{attribute addProperty BoxType "EL6022-0000-0016"}
{attribute addProperty Id "COM_Inputs_ChannelAT %I*ARRAY[0..1] OF COM_Inputs_Channel_DABE08D339849.750COM_Outputs_ChannelAT %Q*ARRAY[0..1] OF COM_Outputs_Channel_60FF225E440550WcStateAT %I*WcState_F855686C1620InfoDataAT %I*InfoData_BC63D37F80100"}
{attribute addProperty CRC "3368682109"}
{attribute addProperty SizeInBites "934"}
{attribute addProperty SizeInBytes "116.75"}
TYPE EL6022_55A24E9B :
STRUCT
	{attribute addProperty Name "COM_Inputs_Channel"}
	COM_Inputs_Channel : ARRAY[0..1] OF COM_Inputs_Channel_DABE08D3;
	{attribute addProperty Name "COM_Outputs_Channel"}
	COM_Outputs_Channel : ARRAY[0..1] OF COM_Outputs_Channel_60FF225E;
	{attribute addProperty Name "WcState"}
	WcState : WcState_F855686C;
	{attribute addProperty Name "InfoData"}
	InfoData : InfoData_BC63D37F;
END_STRUCT
END_TYPE

(* stored: Version 1.2.0.0, ProductVersion 3.1.4024.9
   DUT EL6022_55A24E9B: Id {03cbe744-6259-435f-9984-11165c6c761f} *)
